PROGRAM MAIN
VAR
	bFrontSensor			AT %Q* : BOOL;
	bHomeSensor				AT %Q* : BOOL;
	bRearSensor				AT %Q* : BOOL;
	
	rAnalogSV				AT %I* : REAL;
	
	rAxisPV					AT %Q* : REAL;
	
	bClockwise				AT %I* : BOOL;
	bCounterClockwise		AT %I* : BOOL;
END_VAR

IF rAxisPV > -10 AND rAxisPV < -9 THEN
	bFrontSensor := TRUE;
ELSE
	bFrontSensor := FALSE;
END_IF

IF rAxisPV > 9 AND rAxisPV < 10 THEN
	bHomeSensor := TRUE;
ELSE
	bHomeSensor := FALSE;
END_IF

IF rAxisPV > 59 AND rAxisPV < 60 THEN
	bRearSensor := TRUE;
ELSE
	bRearSensor := FALSE;
END_IF


IF bClockwise THEN
	rAxisPV := rAxisPV - rAnalogSV;
ELSIF bCounterClockwise THEN
	rAxisPV := rAxisPV + rAnalogSV;
END_IF

END_PROGRAM

(* stored: Version 1.1.0.1, ProductVersion 3.1.4024.12
   POU MAIN: Id {769b495a-5390-461e-8f3b-9856b65e90bb}, SpecialFunc None *)
